Yaskawa INFORM job: mataf_small_cylinder_program.JBI

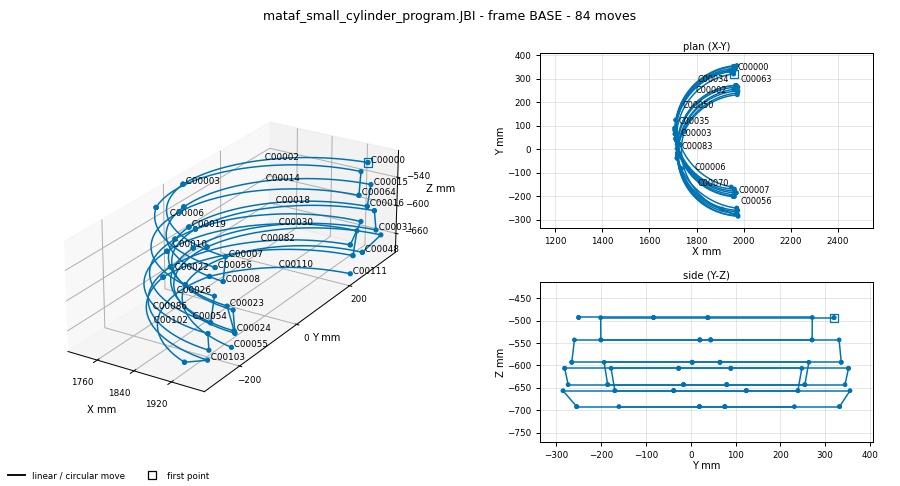
[picture p0: tool path of mataf_small_cylinder_program.JBI in frame BASE, 84 of 122 moves have a stored position in this frame; points joined in program order, loops and branches not executed]
/JOB
//NAME mataf_small_cylinder_program
//POS
///NPOS 112,0,112,0,0,0
///TOOL 0
///POSTYPE BASE
///RECTAN
///RCONF 0,0,0,0,0,0,0,0,0,0,0,0,0,0,0,0,0,0,0,0,0,0,0,0
C00000=1957.478254,319.852640,-493.161500,93.337168,-90.000000,5.000000
C00001=1957.478254,319.852640,-493.161500,93.337168,-90.000000,5.000000
C00002=1777.811898,221.955107,-493.161500,142.989069,-90.000000,5.000000
C00003=1714.501957,38.130693,-493.161500,-171.671404,-90.000000,5.000000
C00004=1714.501957,38.130693,-493.161500,-171.671404,-90.000000,5.000000
C00005=1714.501957,38.130693,-493.161500,-171.671404,-90.000000,5.000000
C00006=1773.821468,-104.660752,-493.161500,-137.639799,-89.999999,5.000000
C00007=1961.271509,-201.221111,-493.161500,-92.158075,-90.000000,5.000000
C00008=1955.524170,-200.712548,-542.798000,-93.350209,-89.999999,5.000000
C00009=1955.524170,-200.712548,-542.798000,-93.350209,-89.999999,5.000000
C00010=1792.548804,-126.436634,-542.798000,-131.539889,-89.999999,5.000000
C00011=1711.565837,44.458571,-542.798000,-173.133664,-89.999999,5.000000
C00012=1711.565837,44.458571,-542.798000,-173.133664,-89.999999,5.000000
C00013=1711.565837,44.458571,-542.798000,-173.133664,-89.999999,5.000000
C00014=1772.683791,234.532145,-542.798000,141.423356,-89.999999,5.000000
C00015=1959.306159,331.273534,-542.798000,92.779492,-90.000000,5.000000
C00016=1949.898370,335.950611,-592.798000,94.792316,-90.000000,5.000000
C00017=1949.898370,335.950611,-592.798000,94.792316,-90.000000,5.000000
C00018=1783.768126,252.836813,-592.798000,136.708890,-90.000000,5.000000
C00019=1708.911793,65.187758,-592.798000,-177.690950,-90.000000,5.000000
C00020=1708.911793,65.187758,-592.798000,-177.690950,-90.000000,5.000000
C00021=1708.911793,65.187758,-592.798000,-177.690950,-90.000000,5.000000
C00022=1791.202777,-118.042587,-592.798000,-132.962130,-90.000000,5.000000
C00023=1959.265353,-193.501079,-592.798000,-92.645961,-89.999999,5.000000
C00024=1968.704572,-185.475076,-642.798000,-90.659079,-89.999999,5.000000
C00025=1968.704572,-185.475076,-642.798000,-90.659079,-89.999999,5.000000
C00026=1789.487109,-109.485781,-642.798000,-134.524908,-90.000000,5.000000
C00027=1708.391799,80.274098,-642.798000,179.023175,-90.000000,5.000000
C00028=1708.391799,80.274098,-642.798000,179.023175,-90.000000,5.000000
C00029=1708.391799,80.274098,-642.798000,179.023175,-90.000000,5.000000
C00030=1785.471900,261.068234,-642.798000,135.147166,-90.000000,5.000000
C00031=1966.164374,344.443054,-642.798000,91.182526,-89.999999,5.000000
C00032=1957.256643,352.172322,-606.195460,-180.000000,-60.000000,-87.006516
C00033=1957.256643,352.172322,-606.195460,-180.000000,-60.000000,-87.006516
C00034=1789.254973,270.033122,-606.195460,180.000000,-60.000000,-46.793208
C00035=1708.039660,89.402312,-606.195460,180.000000,-60.000000,-2.956556
C00036=1708.039660,89.402312,-606.195460,180.000000,-60.000000,-2.956556
C00037=1708.039660,89.402312,-606.195460,180.000000,-60.000000,-2.956556
C00038=1781.217269,-96.248317,-606.195460,180.000000,-60.000000,42.084982
C00039=1962.012701,-178.006120,-606.195460,180.000000,-60.000000,87.811801
C00040=1960.296584,-169.455717,-656.195460,180.000000,-60.000000,87.335391
C00041=1960.296584,-169.455717,-656.195460,180.000000,-60.000000,87.335391
C00042=1763.513368,-69.910529,-656.195460,180.000000,-60.000000,34.984130
C00043=1712.083305,124.016627,-656.195460,180.000000,-60.000000,-10.524164
C00044=1712.083305,124.016627,-656.195460,180.000000,-60.000000,-10.524164
C00045=1712.083305,124.016627,-656.195460,180.000000,-60.000000,-10.524164
C00046=1806.529922,290.057524,-656.195460,180.000000,-60.000000,-52.371886
C00047=1971.451347,355.604936,-656.195460,180.000000,-60.000000,-89.947039
C00048=1943.582822,332.180475,-691.768960,180.000000,-60.000000,-83.739569
C00049=1943.582822,332.180475,-691.768960,180.000000,-60.000000,-83.739569
C00050=1724.057077,160.346276,-691.768960,-180.000000,-60.000000,-18.852633
C00051=1729.523285,19.353131,-691.768960,180.000000,-60.000000,13.116304
C00052=1729.523285,19.353131,-691.768960,180.000000,-60.000000,13.116304
C00053=1729.523285,19.353131,-691.768960,180.000000,-60.000000,13.116304
C00054=1821.468935,-103.130136,-691.768960,180.000000,-60.000000,49.978594
C00055=1947.414881,-160.456727,-691.768960,180.000000,-60.000000,84.128324
C00056=1970.823628,-250.396173,-492.768000,-91.748317,-90.000000,5.000000
C00057=1970.823628,-250.396173,-492.768000,-91.748317,-90.000000,5.000000
C00058=1845.933147,-205.940397,-492.768000,-123.475408,-90.000000,5.000000
C00059=1734.867932,-83.159037,-492.768000,-162.366514,-90.000000,5.000000
C00060=1734.867932,-83.159037,-492.768000,-162.366514,-90.000000,5.000000
C00061=1734.867932,-83.159037,-492.768000,-162.366514,-90.000000,5.000000
C00062=1727.760510,81.156838,-492.768000,160.861694,-90.000000,5.000000
C00063=1969.335735,271.334857,-492.768000,91.850695,-90.000000,5.000000
C00064=1966.184935,270.952002,-542.798000,92.504648,-90.000000,5.000000
C00065=1966.184935,270.952002,-542.798000,92.504648,-90.000000,5.000000
C00066=1797.296853,196.487792,-542.798000,131.822178,-90.000000,5.000000
C00067=1718.146275,20.262581,-542.798000,174.282296,-90.000000,5.000000
C00068=1718.146275,20.262581,-542.798000,174.282296,-90.000000,5.000000
C00069=1718.146275,20.262581,-542.798000,174.282296,-90.000000,5.000000
C00070=1786.351015,-172.728425,-542.798000,-138.984019,-89.999999,5.000000
C00071=1975.114183,-259.719271,-542.798000,-90.716528,-89.999999,5.000000
C00072=1970.775786,-265.730369,-592.798000,-91.655778,-89.999999,5.000000
C00073=1970.775786,-265.730369,-592.798000,-91.655778,-89.999999,5.000000
C00074=1790.943995,-183.983652,-592.798000,-136.433368,-90.000000,5.000000
C00075=1717.978736,3.173467,-592.798000,178.029107,-90.000000,5.000000
C00076=1717.978736,3.173467,-592.798000,178.029107,-90.000000,5.000000
C00077=1717.978736,3.173467,-592.798000,178.029107,-90.000000,5.000000
C00078=1790.048940,182.261336,-592.798000,135.029741,-90.000000,5.000000
C00079=1975.876240,263.645781,-592.798000,90.513285,-89.999999,5.000000
C00080=1958.655084,254.696954,-642.798000,94.310767,-90.000000,5.000000
C00081=1958.655084,254.696954,-642.798000,94.310767,-90.000000,5.000000
C00082=1798.690656,173.735955,-642.798000,135.012602,-90.000000,5.000000
C00083=1719.649537,-16.116226,-642.798000,-177.712441,-90.000000,5.000000
C00084=1719.649537,-16.116226,-642.798000,-177.712441,-90.000000,5.000000
C00085=1719.649537,-16.116226,-642.798000,-177.712441,-90.000000,5.000000
C00086=1790.601374,-190.467499,-642.798000,-135.462442,-90.000000,5.000000
C00087=1972.001142,-273.788720,-642.798000,-91.344228,-90.000000,5.000000
C00088=1975.087910,-281.476883,-606.195460,-180.000000,-60.000000,89.334556
C00089=1975.087910,-281.476883,-606.195460,-180.000000,-60.000000,89.334556
C00090=1789.810139,-201.391658,-606.195460,180.000000,-60.000000,46.063100
C00091=1719.464608,-27.068308,-606.195460,-180.000000,-60.000000,4.701009
C00092=1719.464608,-27.068308,-606.195460,-180.000000,-60.000000,4.701009
C00093=1719.464608,-27.068308,-606.195460,-180.000000,-60.000000,4.701009
C00094=1785.394886,154.308585,-606.195460,180.000000,-60.000000,-39.690921
C00095=1976.406175,247.905365,-606.195460,180.000000,-60.000000,-89.574546
C00096=1973.546314,239.221293,-656.195460,180.000000,-60.000000,-88.890804
C00097=1973.546314,239.221293,-656.195460,180.000000,-60.000000,-88.890804
C00098=1768.940518,119.915510,-656.195460,180.000000,-60.000000,-30.981909
C00099=1717.413077,-38.176269,-656.195460,180.000000,-60.000000,7.077924
C00100=1717.413077,-38.176269,-656.195460,180.000000,-60.000000,7.077924
C00101=1717.413077,-38.176269,-656.195460,180.000000,-60.000000,7.077924
C00102=1807.968476,-213.750872,-656.195460,180.000000,-60.000000,50.683021
C00103=1976.542356,-285.359069,-656.195460,180.000000,-60.000000,89.641844
C00104=1907.722303,-254.667268,-691.915460,180.000000,-60.000000,74.169963
C00105=1907.722303,-254.667268,-691.915460,180.000000,-60.000000,74.169963
C00106=1744.627816,-71.845502,-691.915460,180.000000,-60.000000,15.786688
C00107=1748.184771,76.066762,-691.915460,-180.000000,-60.000000,-19.581077
C00108=1748.184771,76.066762,-691.915460,-180.000000,-60.000000,-19.581077
C00109=1748.184771,76.066762,-691.915460,-180.000000,-60.000000,-19.581077
C00110=1836.206102,180.579442,-691.915460,-180.000000,-60.000000,-52.678082
C00111=1973.009370,231.266096,-691.915460,180.000000,-60.000000,-88.723868
///POSTYPE PULSE
///PULSE
EX00000=92160
EX00001=184320
EX00002=276480
EX00003=368640
///POSTYPE PULSE
///PULSE
EC00000=0
EC00001=0
EC00002=0
EC00003=0
EC00004=0
EC00005=0
EC00006=0
EC00007=0
EC00008=0
EC00009=0
EC00010=0
EC00011=0
EC00012=0
EC00013=0
EC00014=0
EC00015=0
EC00016=0
EC00017=0
EC00018=0
EC00019=0
EC00020=0
EC00021=0
EC00022=0
EC00023=0
EC00024=0
EC00025=0
EC00026=0
EC00027=0
EC00028=0
EC00029=0
EC00030=0
EC00031=0
EC00032=0
EC00033=0
EC00034=0
EC00035=0
EC00036=0
EC00037=0
EC00038=0
EC00039=0
EC00040=0
EC00041=0
EC00042=0
EC00043=0
EC00044=0
EC00045=0
EC00046=0
EC00047=0
EC00048=0
EC00049=0
EC00050=0
EC00051=0
EC00052=0
EC00053=0
EC00054=0
EC00055=0
EC00056=184320
EC00057=184320
EC00058=184320
EC00059=184320
EC00060=184320
EC00061=184320
EC00062=184320
EC00063=184320
EC00064=184320
EC00065=184320
EC00066=184320
EC00067=184320
EC00068=184320
EC00069=184320
EC00070=184320
EC00071=184320
EC00072=184320
EC00073=184320
EC00074=184320
EC00075=184320
EC00076=184320
EC00077=184320
EC00078=184320
EC00079=184320
EC00080=184320
EC00081=184320
EC00082=184320
EC00083=184320
EC00084=184320
EC00085=184320
EC00086=184320
EC00087=184320
EC00088=184320
EC00089=184320
EC00090=184320
EC00091=184320
EC00092=184320
EC00093=184320
EC00094=184320
EC00095=184320
EC00096=184320
EC00097=184320
EC00098=184320
EC00099=184320
EC00100=184320
EC00101=184320
EC00102=184320
EC00103=184320
EC00104=184320
EC00105=184320
EC00106=184320
EC00107=184320
EC00108=184320
EC00109=184320
EC00110=184320
EC00111=184320
//INST
///DATE 2023/07/11 12:06
///ATTR SC,RW,RJ
////FRAME BASE
///GROUP1 RB1,ST1
NOP
MOVJ P009 EX000 VJ=15.00
MOVJ P009 VJ=15.00
MOVJ C00000 EC00000 VJ=15.0
MOVC C00001 EC00001 V=150.0
MOVC C00002 EC00002 V=150.0
MOVC C00003 EC00003 V=150.0
MOVL C00004 EC00004 V=150.0
MOVC C00005 EC00005 V=150.0
MOVC C00006 EC00006 V=150.0
MOVC C00007 EC00007 V=150.0
MOVL C00008 EC00008 V=150.0
MOVC C00009 EC00009 V=150.0
MOVC C00010 EC00010 V=150.0
MOVC C00011 EC00011 V=150.0
MOVL C00012 EC00012 V=150.0
MOVC C00013 EC00013 V=150.0
MOVC C00014 EC00014 V=150.0
MOVC C00015 EC00015 V=150.0
MOVL C00016 EC00016 V=150.0
MOVC C00017 EC00017 V=150.0
MOVC C00018 EC00018 V=150.0
MOVC C00019 EC00019 V=150.0
MOVL C00020 EC00020 V=150.0
MOVC C00021 EC00021 V=150.0
MOVC C00022 EC00022 V=150.0
MOVC C00023 EC00023 V=150.0
MOVL C00024 EC00024 V=150.0
MOVC C00025 EC00025 V=150.0
MOVC C00026 EC00026 V=150.0
MOVC C00027 EC00027 V=150.0
MOVL C00028 EC00028 V=150.0
MOVC C00029 EC00029 V=150.0
MOVC C00030 EC00030 V=150.0
MOVC C00031 EC00031 V=150.0
MOVL C00032 EC00032 V=150.0
MOVC C00033 EC00033 V=150.0
MOVC C00034 EC00034 V=150.0
MOVC C00035 EC00035 V=150.0
MOVL C00036 EC00036 V=150.0
MOVC C00037 EC00037 V=150.0
MOVC C00038 EC00038 V=150.0
MOVC C00039 EC00039 V=150.0
MOVL C00040 EC00040 V=150.0
MOVC C00041 EC00041 V=150.0
MOVC C00042 EC00042 V=150.0
MOVC C00043 EC00043 V=150.0
MOVL C00044 EC00044 V=150.0
MOVC C00045 EC00045 V=150.0
MOVC C00046 EC00046 V=150.0
MOVC C00047 EC00047 V=150.0
MOVL C00048 EC00048 V=150.0
MOVC C00049 EC00049 V=150.0
MOVC C00050 EC00050 V=150.0
MOVC C00051 EC00051 V=150.0
MOVL C00052 EC00052 V=150.0
MOVC C00053 EC00053 V=150.0
MOVC C00054 EC00054 V=150.0
MOVC C00055 EC00055 V=150.0
MOVJ P009 VJ=15.00
MOVL P009 EX00000 V=150.0
MOVJ P009 VJ=15.00
MOVL P009 EX00001 V=150.0
MOVJ C00056 EC00056 VJ=15.0
MOVC C00057 EC00057 V=150.0
MOVC C00058 EC00058 V=150.0
MOVC C00059 EC00059 V=150.0
MOVL C00060 EC00060 V=150.0
MOVC C00061 EC00061 V=150.0
MOVC C00062 EC00062 V=150.0
MOVC C00063 EC00063 V=150.0
MOVL C00064 EC00064 V=150.0
MOVC C00065 EC00065 V=150.0
MOVC C00066 EC00066 V=150.0
MOVC C00067 EC00067 V=150.0
MOVL C00068 EC00068 V=150.0
MOVC C00069 EC00069 V=150.0
MOVC C00070 EC00070 V=150.0
MOVC C00071 EC00071 V=150.0
MOVL C00072 EC00072 V=150.0
MOVC C00073 EC00073 V=150.0
MOVC C00074 EC00074 V=150.0
MOVC C00075 EC00075 V=150.0
MOVL C00076 EC00076 V=150.0
MOVC C00077 EC00077 V=150.0
MOVC C00078 EC00078 V=150.0
MOVC C00079 EC00079 V=150.0
MOVL C00080 EC00080 V=150.0
MOVC C00081 EC00081 V=150.0
MOVC C00082 EC00082 V=150.0
MOVC C00083 EC00083 V=150.0
MOVL C00084 EC00084 V=150.0
MOVC C00085 EC00085 V=150.0
MOVC C00086 EC00086 V=150.0
MOVC C00087 EC00087 V=150.0
MOVL C00088 EC00088 V=150.0
MOVC C00089 EC00089 V=150.0
MOVC C00090 EC00090 V=150.0
MOVC C00091 EC00091 V=150.0
MOVL C00092 EC00092 V=150.0
MOVC C00093 EC00093 V=150.0
MOVC C00094 EC00094 V=150.0
MOVC C00095 EC00095 V=150.0
MOVL C00096 EC00096 V=150.0
MOVC C00097 EC00097 V=150.0
MOVC C00098 EC00098 V=150.0
MOVC C00099 EC00099 V=150.0
MOVL C00100 EC00100 V=150.0
MOVC C00101 EC00101 V=150.0
MOVC C00102 EC00102 V=150.0
MOVC C00103 EC00103 V=150.0
MOVL C00104 EC00104 V=150.0
MOVC C00105 EC00105 V=150.0
MOVC C00106 EC00106 V=150.0
MOVC C00107 EC00107 V=150.0
MOVL C00108 EC00108 V=150.0
MOVC C00109 EC00109 V=150.0
MOVC C00110 EC00110 V=150.0
MOVC C00111 EC00111 V=150.0
MOVJ P009 VJ=15.00
MOVL P009 EX00002 V=150.0
MOVJ P009 VJ=15.00
MOVL P009 EX00003 V=150.0
END
